// TIA Portal V16 export
// export: Created 2021-05-26T11:52:20.6195484Z, ExportSetting WithDefaults, DisplayName Totally Integrated Automation Portal, DisplayVersion V16 Update 4, DisplayName TIA Portal Version Control Interface, DisplayVersion V16 Update 2, DisplayName TIA Portal Openness, DisplayVersion V16 Update 4, DisplayName STEP 7 Professional, DisplayVersion V16 Update 4, DisplayName STEP 7 Safety, DisplayVersion V16, DisplayName WinCC Advanced, DisplayVersion V16 Update 4
DATA_BLOCK "DB_CommCnt_UDP"   // DB41
{ S7_Optimized_Access := 'FALSE' }
VERSION : 0.1
// stored: AutoNumber true, DBAccessibleFromOPCUA true, IsOnlyStoredInLoadMemory false, IsWriteProtectedInAS false
   VAR
      ivBCfast_preCnt : Byte := 16#0F;
      ivBCslow_preCnt : Byte := 16#0F;
      ivDrvCon_preCnt : Byte := 16#0F;
      ivModCon1_preCnt : Byte := 16#0F;
      ivModCon2_preCnt : Byte := 16#0F;
      ivModCon3_preCnt : Byte := 16#0F;
      ivModCon4_preCnt : Byte := 16#0F;
      ivModCon5_preCnt : Byte := 16#0F;
      ivModCon6_preCnt : Byte := 16#0F;
      ivModCon7_preCnt : Byte := 16#0F;
      ivModCon8_preCnt : Byte := 16#0F;
      ivModCon9_preCnt : Byte := 16#0F;
      ivModCon10_preCnt : Byte := 16#0F;
      eBCfast_eComm_act : Bool;
      eBCfast_eComm_det : Bool;
      eBCfast_eComm_trg : Bool;
      stComm_BCfast : Bool;
      eBCslow_eComm_act : Bool;
      eBCslow_eComm_det : Bool;
      eBCslow_eComm_trg : Bool;
      stComm_BCslow : Bool;
      eDrvCon_eComm_act : Bool;
      eDrvCon_eComm_det : Bool;
      eDrvCon_eComm_trg : Bool;
      stComm_DrvCon : Bool;
      eModCon1_eComm_act : Bool;
      eModCon1_eComm_det : Bool;
      eModCon1_eComm_trg : Bool;
      stComm_ModCon1 : Bool;
      eModCon2_eComm_act : Bool;
      eModCon2_eComm_det : Bool;
      eModCon2_eComm_trg : Bool;
      stComm_ModCon2 : Bool;
      eModCon3_eComm_act : Bool;
      eModCon3_eComm_det : Bool;
      eModCon3_eComm_trg : Bool;
      stComm_ModCon3 : Bool;
      eModCon4_eComm_act : Bool;
      eModCon4_eComm_det : Bool;
      eModCon4_eComm_trg : Bool;
      stComm_ModCon4 : Bool;
      eModCon5_eComm_act : Bool;
      eModCon5_eComm_det : Bool;
      eModCon5_eComm_trg : Bool;
      stComm_ModCon5 : Bool;
      eModCon6_eComm_act : Bool;
      eModCon6_eComm_det : Bool;
      eModCon6_eComm_trg : Bool;
      stComm_ModCon6 : Bool;
      eModCon7_eComm_act : Bool;
      eModCon7_eComm_det : Bool;
      eModCon7_eComm_trg : Bool;
      stComm_ModCon7 : Bool;
      eModCon8_eComm_act : Bool;
      eModCon8_eComm_det : Bool;
      eModCon8_eComm_trg : Bool;
      stComm_ModCon8 : Bool;
      eModCon9_eComm_act : Bool;
      eModCon9_eComm_det : Bool;
      eModCon9_eComm_trg : Bool;
      stComm_ModCon9 : Bool;
      eModCon10_eComm_act : Bool;
      eModCon10_eComm_det : Bool;
      eModCon10_eComm_trg : Bool;
      stComm_ModCon10 : Bool;
      res_b19_4 : Bool;
      res_b19_5 : Bool;
      res_b19_6 : Bool;
      res_b19_7 : Bool;
      ivFanCon1_preCnt : Byte := 16#0F;
      ivFanCon2_preCnt : Byte := 16#0F;
      ivFanCon3_preCnt : Byte := 16#0F;
      ivFanCon4_preCnt : Byte := 16#0F;
      eFanCon1_eComm_act : Bool;
      eFanCon1_eComm_det : Bool;
      eFanCon1_eComm_trg : Bool;
      stComm_FanCon1 : Bool;
      eFanCon2_eComm_act : Bool;
      eFanCon2_eComm_det : Bool;
      eFanCon2_eComm_trg : Bool;
      stComm_FanCon2 : Bool;
      eFanCon3_eComm_act : Bool;
      eFanCon3_eComm_det : Bool;
      eFanCon3_eComm_trg : Bool;
      stComm_FanCon3 : Bool;
      eFanCon4_eComm_act : Bool;
      eFanCon4_eComm_det : Bool;
      eFanCon4_eComm_trg : Bool;
      stComm_FanCon4 : Bool;
      ModNum_Cnt : Byte;
   END_VAR
BEGIN
END_DATA_BLOCK
